FUNCTION_BLOCK FB_Operation
VAR_INPUT
	i_bExecute : BOOL; // Flag that indicates the operation should be ran
	i_bCancel : BOOL; // Cancel operation
END_VAR
VAR_OUTPUT
	q_bError : BOOL;
	q_bBusy : BOOL; // Whether the current operation is executing
	q_eCallOp : E_Op := E_Op.NONE; // Signal that another operation should begin executing
	q_sMessage : STRING(EPICS_STRING_SIZE) := 'IDLE'; // Human readable description of the current step
END_VAR
VAR
	eStep : E_OpStep := E_OpStep.IDLE;
	fbTimeoutTimer : TON;
END_VAR
VAR CONSTANT
	STATUS_CHECK_TIMEOUT : TIME := T#30S; // How long the system tries setting the desired state before failing
	VALVE_TIMEOUT : TIME := T#10S; // How long system tries to open or close valve before failing
	ROUGH_CHAMBER_TIMEOUT : TIME := T#5M; // How long to try rough pumping before failing
	TURBO_CHAMBER_TIMEOUT : TIME := T#10M; // How long to try turbo pumping before failing
	PUMP_TIMEOUT : TIME := T#20S; // How long to try to turn on or off pump before failing
END_VAR

q_eCallOp := E_Op.NONE; // Make sure q_eCallOp is cleared before each operation to avoid accidently calling operation again

IF eStep = E_OpStep.IDLE AND i_bExecute = TRUE THEN
	// Start operation
	eStep := E_OpStep.START;
	q_bBusy := TRUE;
	q_bError := FALSE;
END_IF

IF i_bCancel THEN
	M_FatalError('Operation canceled');
END_IF

IF M_TimeoutExpired() THEN // If a timeout has expired, trigger a fatal error
	M_FatalError('Timeout expired');
END_IF

METHOD PROTECTED M_FatalError
VAR_INPUT
	i_ErrorMessage : STRING;
END_VAR
M_ResetTimeoutTimer();
M_SetMessage(i_ErrorMessage);
eStep := E_OpStep.IDLE;
q_bError := TRUE;
q_bBusy := FALSE;
END_METHOD

METHOD PROTECTED M_Finish
VAR_INPUT
END_VAR
M_ResetTimeoutTimer();
eStep := E_OpStep.IDLE;
M_SetMessage('Operation finished');
q_bError := FALSE;
q_bBusy := FALSE;
END_METHOD

METHOD PROTECTED M_ResetTimeoutTimer
VAR_INPUT
END_VAR
fbTimeoutTimer(IN := FALSE);
END_METHOD

METHOD PROTECTED M_RunTimeoutTimer
VAR_INPUT
	i_tTime : TIME; // How long the timer should run before signalling a timeout
END_VAR
fbTimeoutTimer(IN := TRUE, PT := i_tTime);
END_METHOD

METHOD PROTECTED M_SetMessage
VAR_INPUT
	i_sMessage : STRING(EPICS_STRING_SIZE);
END_VAR
q_sMessage := i_sMessage;
END_METHOD

METHOD PROTECTED M_TimeoutExpired : BOOL
VAR_INPUT
END_VAR
fbTimeoutTimer(); // Advance timer
M_TimeoutExpired := fbTimeoutTimer.Q;
END_METHOD

END_FUNCTION_BLOCK

(* stored: Version 1.1.0.1, ProductVersion 3.1.4022.17
   POU FB_Operation: Id {6fc6f593-2545-4a95-82e1-c37424c5cf8b}, SpecialFunc None
   Method M_FatalError: Id {a9657383-9b85-4461-93cb-61ac9678587c}
   Method M_Finish: Id {88ea7fc5-59a3-48a8-88d0-e9fbd7406631}
   Method M_ResetTimeoutTimer: Id {c5848f2a-4ad0-4c43-bb15-e2835c5c0c6d}
   Method M_RunTimeoutTimer: Id {e7e36b84-1348-4c93-80ba-e67778baf763}
   Method M_SetMessage: Id {8436764f-a4c7-4c72-b1be-9a647d3d8896}
   Method M_TimeoutExpired: Id {613a1767-fc71-4068-a0f9-f09d123b2cbd} *)
